# EPICS StreamDevice protocol: poeAdcApp/Db/ADC.proto
ReplyTimeout = 1000;
ReadTimeout  = 1000;
InTerminator = CR LF;

getData {
    separator=', ';
    out "\$1:DATA?";
    in  "[%f]";
}
